(* IEC 61131-3 sources: repolevel_ST_code_completion/output/0121完整版本/repoeval_GreatExampleOfAdvantages/readful_result_history, 2 files *)

(* ---- Home_0.st ---- *)
FUNCTION_BLOCK Home
VAR_INPUT
END_VAR
VAR_OUTPUT
END_VAR
VAR
    GroundFloor: GroundFloor;
    TopFloor: TopFloor;
END_VAR

GroundFloor();
TopFloor();
END_FUNCTION_BLOCK

(* ---- MQTT_STUFF_0.st ---- *)
FUNCTION_BLOCK MQTT_STUFF
VAR_INPUT
END_VAR
VAR_OUTPUT
END_VAR
VAR
    Subscriber: MQTT.MQTTSubscribe;
    init: BOOL;
    InstanceName: CommonTypesAndFunctions.GetInstanceName;
    SubscribeTopic: STRING(255);
    birthTopic: STRING(255);
    found: DINT;
    pt: POINTER TO STRING;
    birthMessage: MQTT.MQTTPublish;
    connectRising: R_TRIG;
    xxx: POINTER TO STRING;
END_VAR

IF NOT init THEN
    init := TRUE;
    Subscriber.SetMqttInOut(MQTT_IN_OUT := GVL_MQTT.MQTT_IN_OUT);
    SubscribeTopic := InstanceName.GetInstanceTopic();
    birthTopic := SubscribeTopic;
    found := CommonTypesAndFunctions.find(str1 := ADR(SubscribeTopic), str2 := ADR('/'));
    found := found + 1 + CommonTypesAndFunctions.find(str1 := ADR(SubscribeTopic[found + 1]), str2 := ADR('/'));
    pt := ADR(SubscribeTopic[found + 1]);
    pt^ := 'Receive/#';
    GVL_MQTT.MQTT_IN_OUT.ClientID := CONCAT('CodesysMqtt', TO_STRING(TICKS.GetTick(xDummy := TRUE)));
END_IF

GVL_MQTT.MQTT_IN_OUT.clientFB(
    MQTT_IN_OUT := GVL_MQTT.MQTT_IN_OUT,
    xConnect := TRUE
);

connectRising(CLK := GVL_MQTT.MQTT_IN_OUT.xConnected);

IF connectRising.Q THEN
    birthMessage.SetMqttInOut(MQTT_IN_OUT := GVL_MQTT.MQTT_IN_OUT);
    birthMessage.Topic := CONCAT(birthTopic, '/Birth');
    birthMessage.Payload := 'Online';
    birthMessage.QoS := 1;
    birthMessage.Retain := TRUE;
    birthMessage.Publish();
    Subscriber.Topic := SubscribeTopic;
    Subscriber.QoS := 1;
    Subscriber.Subscribe();
END_IF
END_FUNCTION_BLOCK
